{attribute 'qualified_only'}
{attribute 'strict'}
TYPE E_CvCraneHandlerType :
(
	eTYPE_UNKNOWN,
	eTYPE_HANDOVER, //Crane Pickup
	eTYPE_TAKEOVER,  //Crane Deposit
	eType_UNDEFINED
);
END_TYPE

(* stored: Version 1.1.0.1, ProductVersion 3.1.4022.12
   DUT E_CvCraneHandlerType: Id {65a75e2c-c487-4dd1-8030-e7c2aace8628} *)
